// TIA Portal V16 export
// export: Created 2021-12-01T20:36:09.36916Z, ExportSetting WithDefaults, DisplayName Totally Integrated Automation Portal, DisplayVersion V16 Update 4, DisplayName TIA Portal Version Control Interface, DisplayVersion V16 Update 2, DisplayName TIA Portal Openness, DisplayVersion V16 Update 4, DisplayName SINAMICS Startdrive Advanced, DisplayVersion V16 Update 5, DisplayName SINAMICS Startdrive G130, G150, S120, S150, SINAMICS MV, S210, DisplayVersion V16 Update 5, DisplayName SINAMICS Startdrive G110M, G120, G120C, G120D, G120P, G115D, DisplayVersion V16 Update 5, DisplayName STEP 7 Professional, DisplayVersion V16 Update 4, DisplayName STEP 7 Safety, DisplayVersion V16, DisplayName WinCC Advanced, DisplayVersion V16 Update 4
FUNCTION "ST00310_FC" : Void   // FC42, LAD
TITLE = ST00310
{ S7_Optimized_Access := 'TRUE' }
VERSION : 0.1
// stored: AutoNumber true, IsIECCheckEnabled false, SetENOAutomatically false, UDAEnableTagReadback false
   VAR_IN_OUT
      OPMODE : "OPMODE_OUT_UDT";
      HMI_EXTENSION : "HMI_EXTENSION_PANEL_UDT";
   END_VAR
   VAR_TEMP
      VDL_TargetPosition : DInt;   // VDL - Target position
      VDL_StartPositioning : Bool;   // VDL - Start auto positioning
      Empty_HS : "RT_HANDSHAKE_UDT";
      PlantIdentifier : WString;
   END_VAR
   VAR CONSTANT
      GetPayloadUID : String := 'ST00310_GP';
   END_VAR
   VAR_TEMP   // added for the SCL form of the ladder/FBD networks
      _w1 : Bool;
      _w2 : Bool;
   END_VAR
BEGIN

REGION Network 1: Alarm
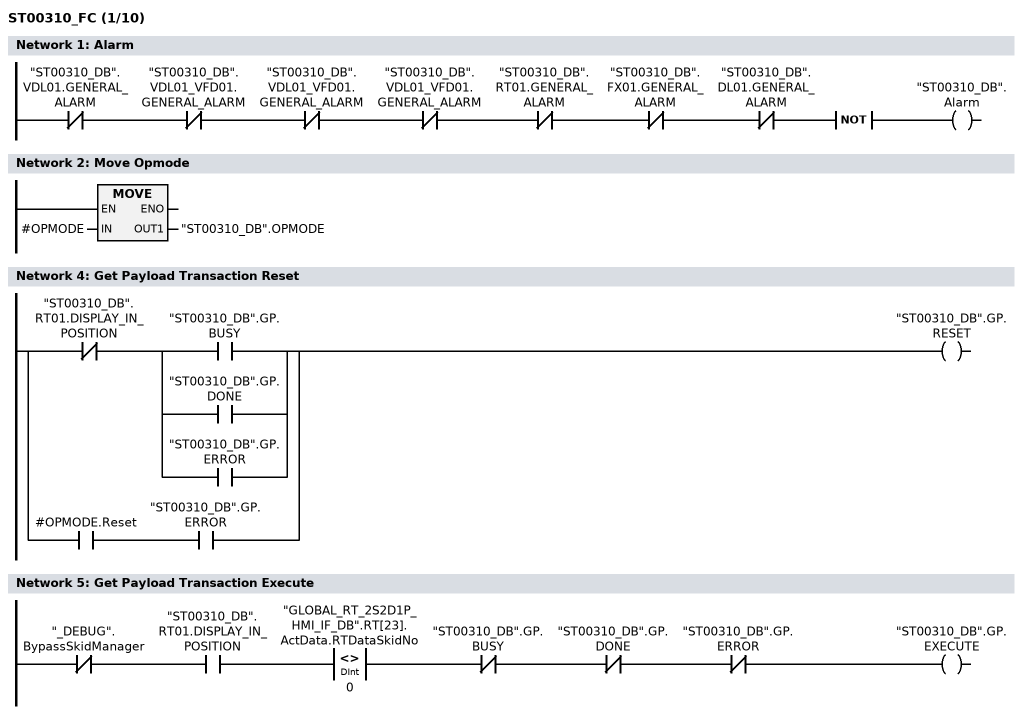
   RUNG wire#powerrail
      I_Contact( "ST00310_DB".VDL01.GENERAL_ALARM )
      I_Contact( "ST00310_DB".VDL01_VFD01.GENERAL_ALARM )
      I_Contact( "ST00310_DB".VDL01_VFD01.GENERAL_ALARM )
      I_Contact( "ST00310_DB".VDL01_VFD01.GENERAL_ALARM )
      I_Contact( "ST00310_DB".RT01.GENERAL_ALARM )
      I_Contact( "ST00310_DB".FX01.GENERAL_ALARM )
      I_Contact( "ST00310_DB".DL01.GENERAL_ALARM )
      Not()
      Coil( "ST00310_DB".Alarm )
   END_RUNG
   // the same network as SCL:
   "ST00310_DB".Alarm := NOT (NOT "ST00310_DB".VDL01.GENERAL_ALARM AND NOT "ST00310_DB".VDL01_VFD01.GENERAL_ALARM AND NOT "ST00310_DB".VDL01_VFD01.GENERAL_ALARM AND NOT "ST00310_DB".VDL01_VFD01.GENERAL_ALARM AND NOT "ST00310_DB".RT01.GENERAL_ALARM AND NOT "ST00310_DB".FX01.GENERAL_ALARM AND NOT "ST00310_DB".DL01.GENERAL_ALARM);
END_REGION

REGION Network 2: Move Opmode
   RUNG wire#powerrail
      Move(in := #OPMODE, out1 => "ST00310_DB".OPMODE)
   END_RUNG
   // the same network as SCL:
   "ST00310_DB".OPMODE := #OPMODE;
END_REGION

REGION Network 3: ==== Get Payload ====
END_REGION

REGION Network 4: Get Payload Transaction Reset
   RUNG wire#powerrail
      I_Contact( "ST00310_DB".RT01.DISPLAY_IN_POSITION )
      wire#w1
      Contact( "ST00310_DB".GP.BUSY )
      wire#w2
      Coil( "ST00310_DB".GP.RESET )
   END_RUNG
   RUNG wire#w1
      Contact( "ST00310_DB".GP.DONE )
   END_RUNG wire#w2
   RUNG wire#w1
      Contact( "ST00310_DB".GP.ERROR )
   END_RUNG wire#w2
   RUNG wire#powerrail
      Contact( #OPMODE.Reset )
      Contact( "ST00310_DB".GP.ERROR )
   END_RUNG wire#w2
   // the same network as SCL:
   "ST00310_DB".GP.RESET := (NOT "ST00310_DB".RT01.DISPLAY_IN_POSITION AND ("ST00310_DB".GP.BUSY OR "ST00310_DB".GP.DONE OR "ST00310_DB".GP.ERROR)) OR (#OPMODE.Reset AND "ST00310_DB".GP.ERROR);
END_REGION

REGION Network 5: Get Payload Transaction Execute
   RUNG wire#powerrail
      I_Contact( "_DEBUG".BypassSkidManager )
      Contact( "ST00310_DB".RT01.DISPLAY_IN_POSITION )
      { S7_Templates := "SrcType := DInt" } NE_Contact(in1 := "GLOBAL_RT_2S2D1P_HMI_IF_DB".RT[23].ActData.RTDataSkidNo, in2 := 0)
      I_Contact( "ST00310_DB".GP.BUSY )
      I_Contact( "ST00310_DB".GP.DONE )
      I_Contact( "ST00310_DB".GP.ERROR )
      Coil( "ST00310_DB".GP.EXECUTE )
   END_RUNG
   // the same network as SCL:
   "ST00310_DB".GP.EXECUTE := NOT "_DEBUG".BypassSkidManager AND "ST00310_DB".RT01.DISPLAY_IN_POSITION AND ("GLOBAL_RT_2S2D1P_HMI_IF_DB".RT[23].ActData.RTDataSkidNo <> 0) AND NOT "ST00310_DB".GP.BUSY AND NOT "ST00310_DB".GP.DONE AND NOT "ST00310_DB".GP.ERROR;
END_REGION

REGION Network 6: Get Payload Transaction Control
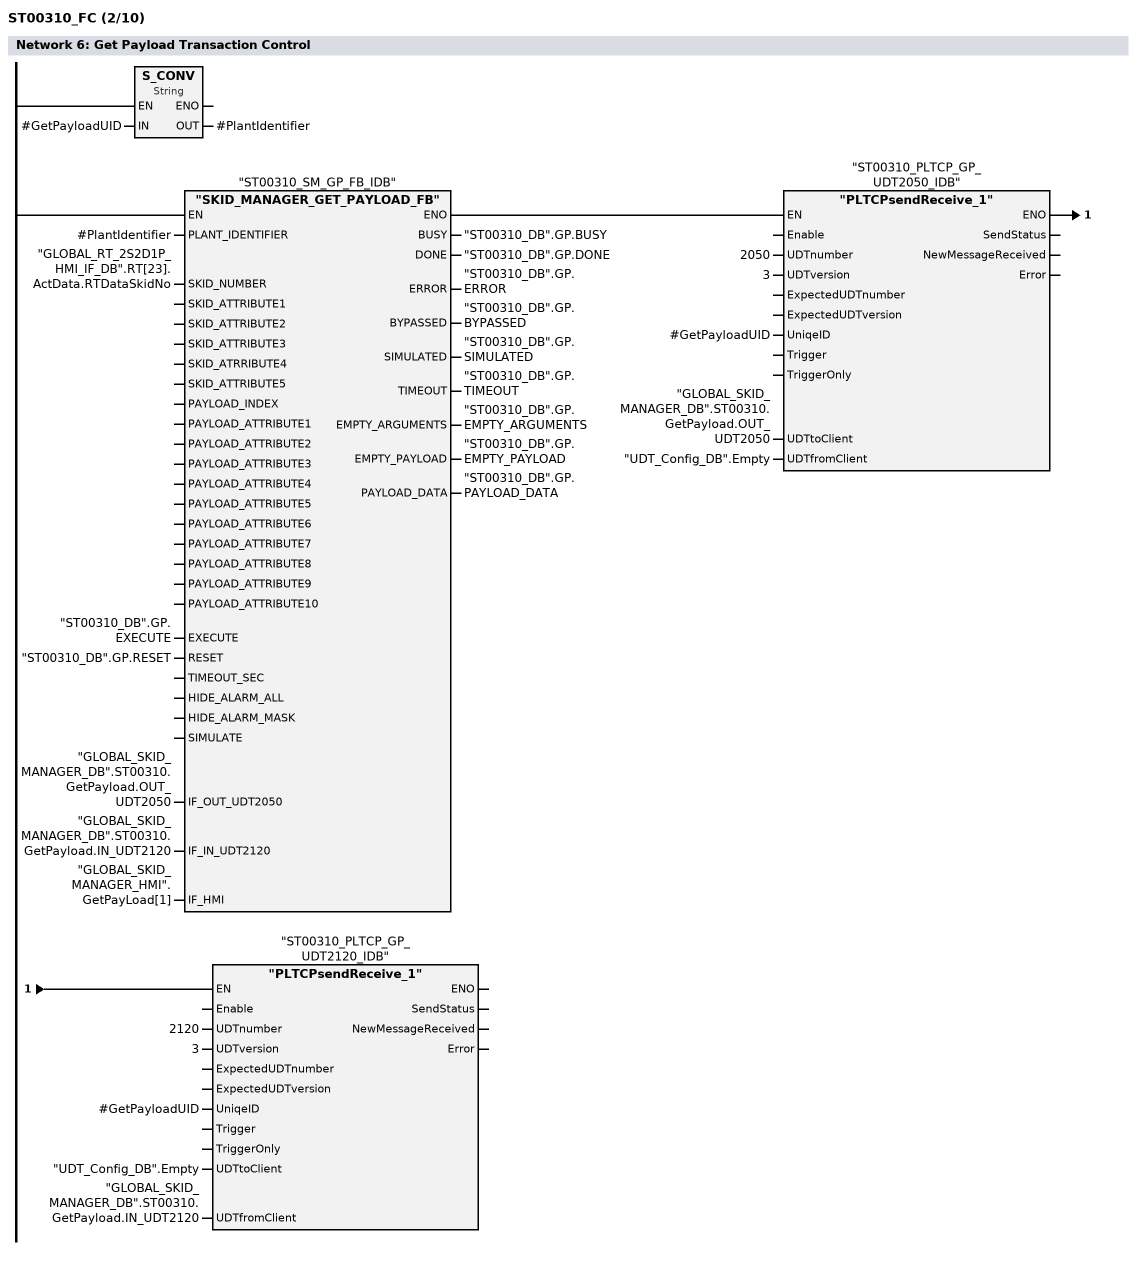
   RUNG wire#powerrail
      { S7_Templates := "[src_type := String, dest_type := WString]" } S_CONV(IN := #GetPayloadUID, OUT => #PlantIdentifier)
   END_RUNG
   RUNG wire#powerrail
      "ST00310_SM_GP_FB_IDB"(PLANT_IDENTIFIER := #PlantIdentifier, SKID_NUMBER := "GLOBAL_RT_2S2D1P_HMI_IF_DB".RT[23].ActData.RTDataSkidNo, SKID_ATTRIBUTE1 :=, SKID_ATTRIBUTE2 :=, SKID_ATTRIBUTE3 :=, SKID_ATRRIBUTE4 :=, SKID_ATTRIBUTE5 :=, PAYLOAD_INDEX :=, PAYLOAD_ATTRIBUTE1 :=, PAYLOAD_ATTRIBUTE2 :=, PAYLOAD_ATTRIBUTE3 :=, PAYLOAD_ATTRIBUTE4 :=, PAYLOAD_ATTRIBUTE5 :=, PAYLOAD_ATTRIBUTE6 :=, PAYLOAD_ATTRIBUTE7 :=, PAYLOAD_ATTRIBUTE8 :=, PAYLOAD_ATTRIBUTE9 :=, PAYLOAD_ATTRIBUTE10 :=, EXECUTE := "ST00310_DB".GP.EXECUTE, RESET := "ST00310_DB".GP.RESET, TIMEOUT_SEC :=, HIDE_ALARM_ALL :=, HIDE_ALARM_MASK :=, SIMULATE :=, IF_OUT_UDT2050 := "GLOBAL_SKID_MANAGER_DB".ST00310.GetPayload.OUT_UDT2050, IF_IN_UDT2120 := "GLOBAL_SKID_MANAGER_DB".ST00310.GetPayload.IN_UDT2120, IF_HMI := "GLOBAL_SKID_MANAGER_HMI".GetPayLoad[1], BUSY => "ST00310_DB".GP.BUSY, DONE => "ST00310_DB".GP.DONE, ERROR => "ST00310_DB".GP.ERROR, BYPASSED => "ST00310_DB".GP.BYPASSED, SIMULATED => "ST00310_DB".GP.SIMULATED, TIMEOUT => "ST00310_DB".GP.TIMEOUT, EMPTY_ARGUMENTS => "ST00310_DB".GP.EMPTY_ARGUMENTS, EMPTY_PAYLOAD => "ST00310_DB".GP.EMPTY_PAYLOAD, PAYLOAD_DATA => "ST00310_DB".GP.PAYLOAD_DATA)
      "ST00310_PLTCP_GP_UDT2050_IDB"(Enable :=, UDTnumber := 2050, UDTversion := 3, ExpectedUDTnumber :=, ExpectedUDTversion :=, UniqeID := #GetPayloadUID, Trigger :=, TriggerOnly :=, UDTtoClient := "GLOBAL_SKID_MANAGER_DB".ST00310.GetPayload.OUT_UDT2050, UDTfromClient := "UDT_Config_DB".Empty, SendStatus =>, NewMessageReceived =>, Error =>)
      "ST00310_PLTCP_GP_UDT2120_IDB"(Enable :=, UDTnumber := 2120, UDTversion := 3, ExpectedUDTnumber :=, ExpectedUDTversion :=, UniqeID := #GetPayloadUID, Trigger :=, TriggerOnly :=, UDTtoClient := "UDT_Config_DB".Empty, UDTfromClient := "GLOBAL_SKID_MANAGER_DB".ST00310.GetPayload.IN_UDT2120, SendStatus =>, NewMessageReceived =>, Error =>)
   END_RUNG
   // the same network as SCL:
   S_CONV(IN := #GetPayloadUID, OUT => #PlantIdentifier);
   "ST00310_SM_GP_FB_IDB"(PLANT_IDENTIFIER := #PlantIdentifier,   // "SKID_MANAGER_GET_PAYLOAD_FB"
                          SKID_NUMBER := "GLOBAL_RT_2S2D1P_HMI_IF_DB".RT[23].ActData.RTDataSkidNo,
                          EXECUTE := "ST00310_DB".GP.EXECUTE,
                          RESET := "ST00310_DB".GP.RESET,
                          IF_OUT_UDT2050 := "GLOBAL_SKID_MANAGER_DB".ST00310.GetPayload.OUT_UDT2050,
                          IF_IN_UDT2120 := "GLOBAL_SKID_MANAGER_DB".ST00310.GetPayload.IN_UDT2120,
                          IF_HMI := "GLOBAL_SKID_MANAGER_HMI".GetPayLoad[1],
                          BUSY => "ST00310_DB".GP.BUSY,
                          DONE => "ST00310_DB".GP.DONE,
                          ERROR => "ST00310_DB".GP.ERROR,
                          BYPASSED => "ST00310_DB".GP.BYPASSED,
                          SIMULATED => "ST00310_DB".GP.SIMULATED,
                          TIMEOUT => "ST00310_DB".GP.TIMEOUT,
                          EMPTY_ARGUMENTS => "ST00310_DB".GP.EMPTY_ARGUMENTS,
                          EMPTY_PAYLOAD => "ST00310_DB".GP.EMPTY_PAYLOAD,
                          PAYLOAD_DATA => "ST00310_DB".GP.PAYLOAD_DATA,
                          ENO => #_w1);
   "ST00310_PLTCP_GP_UDT2050_IDB"(EN := #_w1,   // "PLTCPsendReceive_1"
                           UDTnumber := 2050,
                           UDTversion := 3,
                           UniqeID := #GetPayloadUID,
                           UDTtoClient := "GLOBAL_SKID_MANAGER_DB".ST00310.GetPayload.OUT_UDT2050,
                           UDTfromClient := "UDT_Config_DB".Empty,
                           ENO => #_w2);
   IF #_w2 THEN
       "ST00310_PLTCP_GP_UDT2120_IDB"(UDTnumber := 2120,   // "PLTCPsendReceive_1"
                               UDTversion := 3,
                               UniqeID := #GetPayloadUID,
                               UDTtoClient := "UDT_Config_DB".Empty,
                               UDTfromClient := "GLOBAL_SKID_MANAGER_DB".ST00310.GetPayload.IN_UDT2120);
   END_IF;
END_REGION

REGION Network 7: *******************VDL01 Control*******************
END_REGION

REGION Network 8 (SCL): VDL01 Parameters


   "ST00310_DB".VDL01.PARA_SET.Para.StopNextPos := true;
   "ST00310_DB".VDL01.PARA_SET.Set.DistPos := 10;
   "ST00310_DB".VDL01.PARA_SET.Set.DistSDFwd := 550;
   "ST00310_DB".VDL01.PARA_SET.Set.DistSDRev := 550;
   "ST00310_DB".VDL01.PARA_SET.Set.DistStopFwd := 20;
   "ST00310_DB".VDL01.PARA_SET.Set.DistStopRev := 20;
   "ST00310_DB".VDL01.PARA_SET.Set.EncValFac := 1;
   "ST00310_DB".VDL01.PARA_SET.Set.LastPos := 2;
   "ST00310_DB".VDL01.PARA_SET.Set.LimSwSWFwd := 9130;
   "ST00310_DB".VDL01.PARA_SET.Set.LimSwSWRev := 550;


   "ST00310_DB".VDL01.PARA_SET.Set.Pos1S := 590;
   "ST00310_DB".VDL01.PARA_SET.Set.Pos2S := 9115;

   "ST00310_DB".VDL01.PARA_SET.Set.RtPos1Pos2 := 300;
END_REGION

REGION Network 9: VDL01 Distance Meter
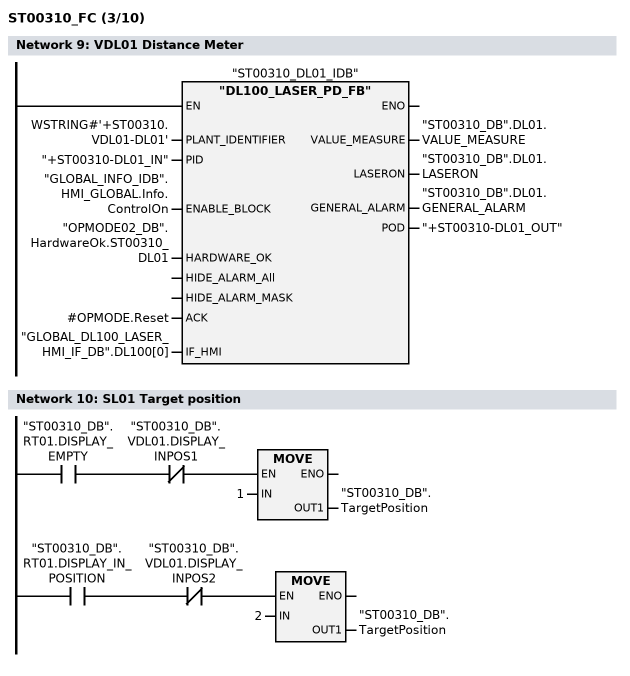
   RUNG wire#powerrail
      "ST00310_DL01_IDB"(PLANT_IDENTIFIER := WSTRING#'+ST00310.VDL01-DL01', PID := "+ST00310-DL01_IN", ENABLE_BLOCK := "GLOBAL_INFO_IDB".HMI_GLOBAL.Info.ControlOn, HARDWARE_OK := "OPMODE02_DB".HardwareOk.ST00310_DL01, HIDE_ALARM_All :=, HIDE_ALARM_MASK :=, ACK := #OPMODE.Reset, IF_HMI := "GLOBAL_DL100_LASER_HMI_IF_DB".DL100[0], VALUE_MEASURE => "ST00310_DB".DL01.VALUE_MEASURE, LASERON => "ST00310_DB".DL01.LASERON, GENERAL_ALARM => "ST00310_DB".DL01.GENERAL_ALARM, POD => "+ST00310-DL01_OUT")
   END_RUNG
   // the same network as SCL:
   "ST00310_DL01_IDB"(PLANT_IDENTIFIER := WSTRING#'+ST00310.VDL01-DL01',   // "DL100_LASER_PD_FB"
                      PID := "+ST00310-DL01_IN",
                      ENABLE_BLOCK := "GLOBAL_INFO_IDB".HMI_GLOBAL.Info.ControlOn,
                      HARDWARE_OK := "OPMODE02_DB".HardwareOk.ST00310_DL01,
                      ACK := #OPMODE.Reset,
                      IF_HMI := "GLOBAL_DL100_LASER_HMI_IF_DB".DL100[0],
                      VALUE_MEASURE => "ST00310_DB".DL01.VALUE_MEASURE,
                      LASERON => "ST00310_DB".DL01.LASERON,
                      GENERAL_ALARM => "ST00310_DB".DL01.GENERAL_ALARM,
                      POD => "+ST00310-DL01_OUT");
END_REGION

REGION Network 10: SL01 Target position
   RUNG wire#powerrail
      Contact( "ST00310_DB".RT01.DISPLAY_EMPTY )
      I_Contact( "ST00310_DB".VDL01.DISPLAY_INPOS1 )
      Move(in := 1, out1 => "ST00310_DB".TargetPosition)
   END_RUNG
   RUNG wire#powerrail
      Contact( "ST00310_DB".RT01.DISPLAY_IN_POSITION )
      I_Contact( "ST00310_DB".VDL01.DISPLAY_INPOS2 )
      Move(in := 2, out1 => "ST00310_DB".TargetPosition)
   END_RUNG
   // the same network as SCL:
   IF "ST00310_DB".RT01.DISPLAY_EMPTY AND NOT "ST00310_DB".VDL01.DISPLAY_INPOS1 THEN
       "ST00310_DB".TargetPosition := 1;
   END_IF;
   IF "ST00310_DB".RT01.DISPLAY_IN_POSITION AND NOT "ST00310_DB".VDL01.DISPLAY_INPOS2 THEN
       "ST00310_DB".TargetPosition := 2;
   END_IF;
END_REGION

REGION Network 11: VDL01 FB Control
   // 1. RT occupied -> go to 8,5m
   // 2. RT not occupied -> go to 0m
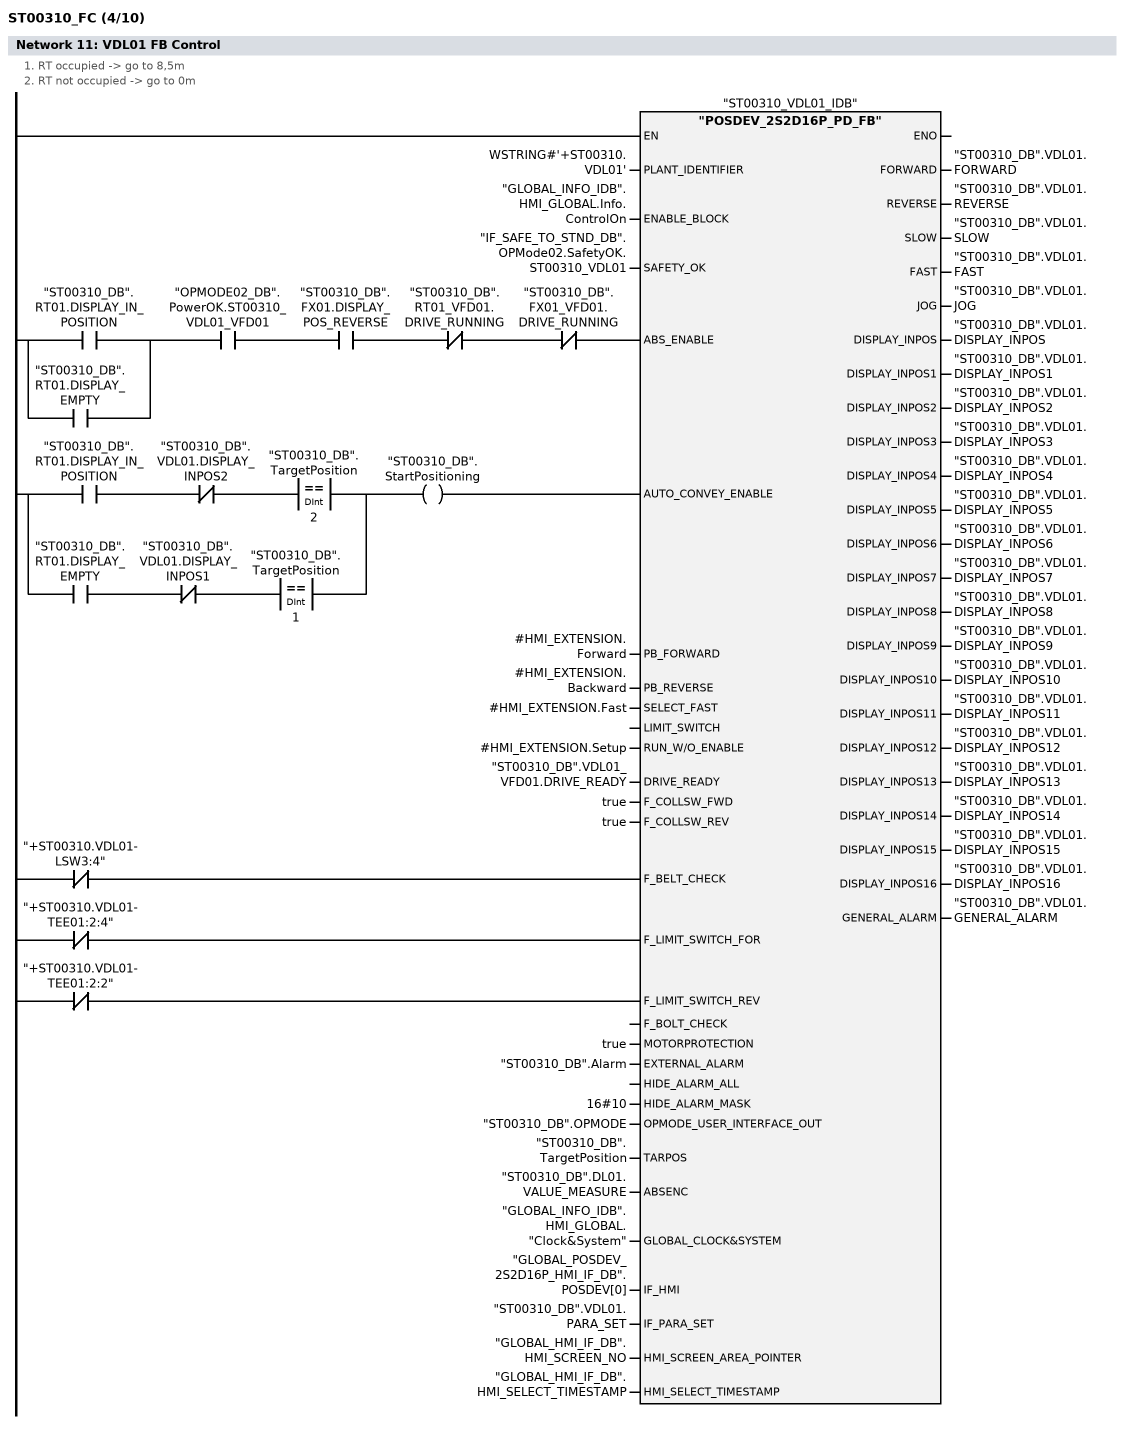
   RUNG wire#powerrail
      "ST00310_VDL01_IDB"(ABS_ENABLE := wire#w2, AUTO_CONVEY_ENABLE := wire#w4, F_BELT_CHECK := wire#w5, F_LIMIT_SWITCH_FOR := wire#w6, F_LIMIT_SWITCH_REV := wire#w7, PLANT_IDENTIFIER := WSTRING#'+ST00310.VDL01', ENABLE_BLOCK := "GLOBAL_INFO_IDB".HMI_GLOBAL.Info.ControlOn, SAFETY_OK := "IF_SAFE_TO_STND_DB".OPMode02.SafetyOK.ST00310_VDL01, PB_FORWARD := #HMI_EXTENSION.Forward, PB_REVERSE := #HMI_EXTENSION.Backward, SELECT_FAST := #HMI_EXTENSION.Fast, LIMIT_SWITCH :=, "RUN_W/O_ENABLE" := #HMI_EXTENSION.Setup, DRIVE_READY := "ST00310_DB".VDL01_VFD01.DRIVE_READY, F_COLLSW_FWD := true, F_COLLSW_REV := true, F_BOLT_CHECK :=, MOTORPROTECTION := true, EXTERNAL_ALARM := "ST00310_DB".Alarm, HIDE_ALARM_ALL :=, HIDE_ALARM_MASK := 16#10, OPMODE_USER_INTERFACE_OUT := "ST00310_DB".OPMODE, TARPOS := "ST00310_DB".TargetPosition, ABSENC := "ST00310_DB".DL01.VALUE_MEASURE, "GLOBAL_CLOCK&SYSTEM" := "GLOBAL_INFO_IDB".HMI_GLOBAL."Clock&System", IF_HMI := "GLOBAL_POSDEV_2S2D16P_HMI_IF_DB".POSDEV[0], IF_PARA_SET := "ST00310_DB".VDL01.PARA_SET, HMI_SCREEN_AREA_POINTER := "GLOBAL_HMI_IF_DB".HMI_SCREEN_NO, HMI_SELECT_TIMESTAMP := "GLOBAL_HMI_IF_DB".HMI_SELECT_TIMESTAMP, FORWARD => "ST00310_DB".VDL01.FORWARD, REVERSE => "ST00310_DB".VDL01.REVERSE, SLOW => "ST00310_DB".VDL01.SLOW, FAST => "ST00310_DB".VDL01.FAST, JOG => "ST00310_DB".VDL01.JOG, DISPLAY_INPOS => "ST00310_DB".VDL01.DISPLAY_INPOS, DISPLAY_INPOS1 => "ST00310_DB".VDL01.DISPLAY_INPOS1, DISPLAY_INPOS2 => "ST00310_DB".VDL01.DISPLAY_INPOS2, DISPLAY_INPOS3 => "ST00310_DB".VDL01.DISPLAY_INPOS3, DISPLAY_INPOS4 => "ST00310_DB".VDL01.DISPLAY_INPOS4, DISPLAY_INPOS5 => "ST00310_DB".VDL01.DISPLAY_INPOS5, DISPLAY_INPOS6 => "ST00310_DB".VDL01.DISPLAY_INPOS6, DISPLAY_INPOS7 => "ST00310_DB".VDL01.DISPLAY_INPOS7, DISPLAY_INPOS8 => "ST00310_DB".VDL01.DISPLAY_INPOS8, DISPLAY_INPOS9 => "ST00310_DB".VDL01.DISPLAY_INPOS9, DISPLAY_INPOS10 => "ST00310_DB".VDL01.DISPLAY_INPOS10, DISPLAY_INPOS11 => "ST00310_DB".VDL01.DISPLAY_INPOS11, DISPLAY_INPOS12 => "ST00310_DB".VDL01.DISPLAY_INPOS12, DISPLAY_INPOS13 => "ST00310_DB".VDL01.DISPLAY_INPOS13, DISPLAY_INPOS14 => "ST00310_DB".VDL01.DISPLAY_INPOS14, DISPLAY_INPOS15 => "ST00310_DB".VDL01.DISPLAY_INPOS15, DISPLAY_INPOS16 => "ST00310_DB".VDL01.DISPLAY_INPOS16, GENERAL_ALARM => "ST00310_DB".VDL01.GENERAL_ALARM)
   END_RUNG
   RUNG wire#powerrail
      Contact( "ST00310_DB".RT01.DISPLAY_IN_POSITION )
      wire#w1
      Contact( "OPMODE02_DB".PowerOK.ST00310_VDL01_VFD01 )
      Contact( "ST00310_DB".FX01.DISPLAY_POS_REVERSE )
      I_Contact( "ST00310_DB".RT01_VFD01.DRIVE_RUNNING )
      I_Contact( "ST00310_DB".FX01_VFD01.DRIVE_RUNNING )
   END_RUNG wire#w2
   RUNG wire#powerrail
      Contact( "ST00310_DB".RT01.DISPLAY_EMPTY )
   END_RUNG wire#w1
   RUNG wire#powerrail
      Contact( "ST00310_DB".RT01.DISPLAY_IN_POSITION )
      I_Contact( "ST00310_DB".VDL01.DISPLAY_INPOS2 )
      { S7_Templates := "SrcType := DInt" } EQ_Contact(in1 := "ST00310_DB".TargetPosition, in2 := 2)
      wire#w3
      Coil( "ST00310_DB".StartPositioning )
   END_RUNG wire#w4
   RUNG wire#powerrail
      Contact( "ST00310_DB".RT01.DISPLAY_EMPTY )
      I_Contact( "ST00310_DB".VDL01.DISPLAY_INPOS1 )
      { S7_Templates := "SrcType := DInt" } EQ_Contact(in1 := "ST00310_DB".TargetPosition, in2 := 1)
   END_RUNG wire#w3
   RUNG wire#powerrail
      I_Contact( "+ST00310.VDL01-LSW3:4" )
   END_RUNG wire#w5
   RUNG wire#powerrail
      I_Contact( "+ST00310.VDL01-TEE01:2:4" )
   END_RUNG wire#w6
   RUNG wire#powerrail
      I_Contact( "+ST00310.VDL01-TEE01:2:2" )
   END_RUNG wire#w7
   // the same network as SCL:
   "ST00310_DB".StartPositioning := ("ST00310_DB".RT01.DISPLAY_IN_POSITION AND NOT "ST00310_DB".VDL01.DISPLAY_INPOS2 AND ("ST00310_DB".TargetPosition = 2)) OR ("ST00310_DB".RT01.DISPLAY_EMPTY AND NOT "ST00310_DB".VDL01.DISPLAY_INPOS1 AND ("ST00310_DB".TargetPosition = 1));
   "ST00310_VDL01_IDB"(PLANT_IDENTIFIER := WSTRING#'+ST00310.VDL01',   // "POSDEV_2S2D16P_PD_FB"
                       ENABLE_BLOCK := "GLOBAL_INFO_IDB".HMI_GLOBAL.Info.ControlOn,
                       SAFETY_OK := "IF_SAFE_TO_STND_DB".OPMode02.SafetyOK.ST00310_VDL01,
                       ABS_ENABLE := ("ST00310_DB".RT01.DISPLAY_IN_POSITION OR "ST00310_DB".RT01.DISPLAY_EMPTY) AND "OPMODE02_DB".PowerOK.ST00310_VDL01_VFD01 AND "ST00310_DB".FX01.DISPLAY_POS_REVERSE AND NOT "ST00310_DB".RT01_VFD01.DRIVE_RUNNING AND NOT "ST00310_DB".FX01_VFD01.DRIVE_RUNNING,
                       AUTO_CONVEY_ENABLE := "ST00310_DB".StartPositioning,
                       PB_FORWARD := #HMI_EXTENSION.Forward,
                       PB_REVERSE := #HMI_EXTENSION.Backward,
                       SELECT_FAST := #HMI_EXTENSION.Fast,
                       "RUN_W/O_ENABLE" := #HMI_EXTENSION.Setup,
                       DRIVE_READY := "ST00310_DB".VDL01_VFD01.DRIVE_READY,
                       F_COLLSW_FWD := true,
                       F_COLLSW_REV := true,
                       F_BELT_CHECK := NOT "+ST00310.VDL01-LSW3:4",
                       F_LIMIT_SWITCH_FOR := NOT "+ST00310.VDL01-TEE01:2:4",
                       F_LIMIT_SWITCH_REV := NOT "+ST00310.VDL01-TEE01:2:2",
                       MOTORPROTECTION := true,
                       EXTERNAL_ALARM := "ST00310_DB".Alarm,
                       HIDE_ALARM_MASK := 16#10,
                       OPMODE_USER_INTERFACE_OUT := "ST00310_DB".OPMODE,
                       TARPOS := "ST00310_DB".TargetPosition,
                       ABSENC := "ST00310_DB".DL01.VALUE_MEASURE,
                       "GLOBAL_CLOCK&SYSTEM" := "GLOBAL_INFO_IDB".HMI_GLOBAL."Clock&System",
                       IF_HMI := "GLOBAL_POSDEV_2S2D16P_HMI_IF_DB".POSDEV[0],
                       IF_PARA_SET := "ST00310_DB".VDL01.PARA_SET,
                       HMI_SCREEN_AREA_POINTER := "GLOBAL_HMI_IF_DB".HMI_SCREEN_NO,
                       HMI_SELECT_TIMESTAMP := "GLOBAL_HMI_IF_DB".HMI_SELECT_TIMESTAMP,
                       FORWARD => "ST00310_DB".VDL01.FORWARD,
                       REVERSE => "ST00310_DB".VDL01.REVERSE,
                       SLOW => "ST00310_DB".VDL01.SLOW,
                       FAST => "ST00310_DB".VDL01.FAST,
                       JOG => "ST00310_DB".VDL01.JOG,
                       DISPLAY_INPOS => "ST00310_DB".VDL01.DISPLAY_INPOS,
                       DISPLAY_INPOS1 => "ST00310_DB".VDL01.DISPLAY_INPOS1,
                       DISPLAY_INPOS2 => "ST00310_DB".VDL01.DISPLAY_INPOS2,
                       DISPLAY_INPOS3 => "ST00310_DB".VDL01.DISPLAY_INPOS3,
                       DISPLAY_INPOS4 => "ST00310_DB".VDL01.DISPLAY_INPOS4,
                       DISPLAY_INPOS5 => "ST00310_DB".VDL01.DISPLAY_INPOS5,
                       DISPLAY_INPOS6 => "ST00310_DB".VDL01.DISPLAY_INPOS6,
                       DISPLAY_INPOS7 => "ST00310_DB".VDL01.DISPLAY_INPOS7,
                       DISPLAY_INPOS8 => "ST00310_DB".VDL01.DISPLAY_INPOS8,
                       DISPLAY_INPOS9 => "ST00310_DB".VDL01.DISPLAY_INPOS9,
                       DISPLAY_INPOS10 => "ST00310_DB".VDL01.DISPLAY_INPOS10,
                       DISPLAY_INPOS11 => "ST00310_DB".VDL01.DISPLAY_INPOS11,
                       DISPLAY_INPOS12 => "ST00310_DB".VDL01.DISPLAY_INPOS12,
                       DISPLAY_INPOS13 => "ST00310_DB".VDL01.DISPLAY_INPOS13,
                       DISPLAY_INPOS14 => "ST00310_DB".VDL01.DISPLAY_INPOS14,
                       DISPLAY_INPOS15 => "ST00310_DB".VDL01.DISPLAY_INPOS15,
                       DISPLAY_INPOS16 => "ST00310_DB".VDL01.DISPLAY_INPOS16,
                       GENERAL_ALARM => "ST00310_DB".VDL01.GENERAL_ALARM);
END_REGION

REGION Network 12: VDL01 Speed
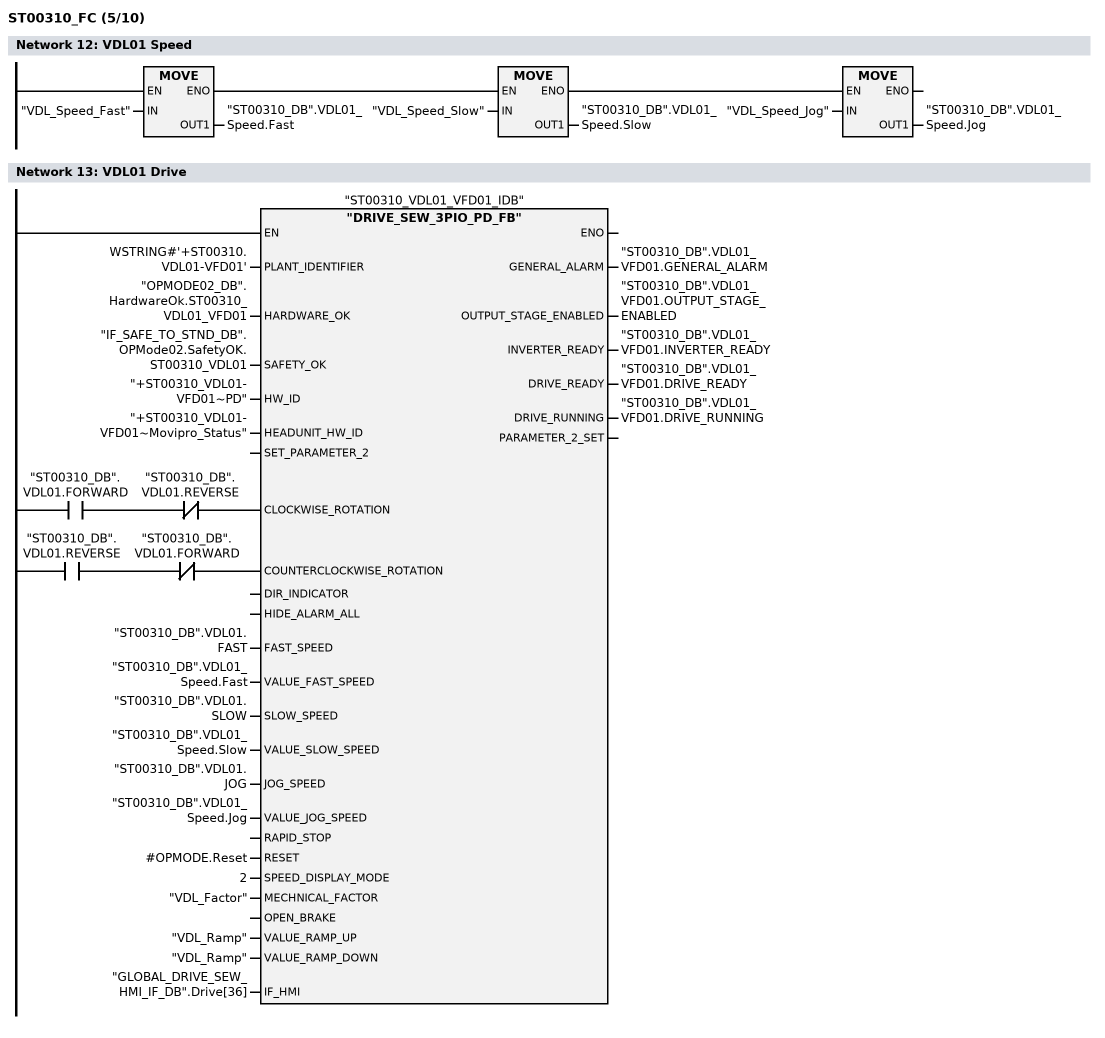
   RUNG wire#powerrail
      Move(in := "VDL_Speed_Fast", out1 => "ST00310_DB".VDL01_Speed.Fast)
      Move(in := "VDL_Speed_Slow", out1 => "ST00310_DB".VDL01_Speed.Slow)
      Move(in := "VDL_Speed_Jog", out1 => "ST00310_DB".VDL01_Speed.Jog)
   END_RUNG
   // the same network as SCL:
   "ST00310_DB".VDL01_Speed.Fast := "VDL_Speed_Fast";
   "ST00310_DB".VDL01_Speed.Slow := "VDL_Speed_Slow";
   "ST00310_DB".VDL01_Speed.Jog := "VDL_Speed_Jog";
END_REGION

REGION Network 13: VDL01 Drive
   RUNG wire#powerrail
      "ST00310_VDL01_VFD01_IDB"(CLOCKWISE_ROTATION := wire#w1, COUNTERCLOCKWISE_ROTATION := wire#w2, PLANT_IDENTIFIER := WSTRING#'+ST00310.VDL01-VFD01', HARDWARE_OK := "OPMODE02_DB".HardwareOk.ST00310_VDL01_VFD01, SAFETY_OK := "IF_SAFE_TO_STND_DB".OPMode02.SafetyOK.ST00310_VDL01, HW_ID := "+ST00310_VDL01-VFD01~PD", HEADUNIT_HW_ID := "+ST00310_VDL01-VFD01~Movipro_Status", SET_PARAMETER_2 :=, DIR_INDICATOR :=, HIDE_ALARM_ALL :=, FAST_SPEED := "ST00310_DB".VDL01.FAST, VALUE_FAST_SPEED := "ST00310_DB".VDL01_Speed.Fast, SLOW_SPEED := "ST00310_DB".VDL01.SLOW, VALUE_SLOW_SPEED := "ST00310_DB".VDL01_Speed.Slow, JOG_SPEED := "ST00310_DB".VDL01.JOG, VALUE_JOG_SPEED := "ST00310_DB".VDL01_Speed.Jog, RAPID_STOP :=, RESET := #OPMODE.Reset, SPEED_DISPLAY_MODE := 2, MECHNICAL_FACTOR := "VDL_Factor", OPEN_BRAKE :=, VALUE_RAMP_UP := "VDL_Ramp", VALUE_RAMP_DOWN := "VDL_Ramp", IF_HMI := "GLOBAL_DRIVE_SEW_HMI_IF_DB".Drive[36], GENERAL_ALARM => "ST00310_DB".VDL01_VFD01.GENERAL_ALARM, OUTPUT_STAGE_ENABLED => "ST00310_DB".VDL01_VFD01.OUTPUT_STAGE_ENABLED, INVERTER_READY => "ST00310_DB".VDL01_VFD01.INVERTER_READY, DRIVE_READY => "ST00310_DB".VDL01_VFD01.DRIVE_READY, DRIVE_RUNNING => "ST00310_DB".VDL01_VFD01.DRIVE_RUNNING, PARAMETER_2_SET =>)
   END_RUNG
   RUNG wire#powerrail
      Contact( "ST00310_DB".VDL01.FORWARD )
      I_Contact( "ST00310_DB".VDL01.REVERSE )
   END_RUNG wire#w1
   RUNG wire#powerrail
      Contact( "ST00310_DB".VDL01.REVERSE )
      I_Contact( "ST00310_DB".VDL01.FORWARD )
   END_RUNG wire#w2
   // the same network as SCL:
   "ST00310_VDL01_VFD01_IDB"(PLANT_IDENTIFIER := WSTRING#'+ST00310.VDL01-VFD01',   // "DRIVE_SEW_3PIO_PD_FB"
                           HARDWARE_OK := "OPMODE02_DB".HardwareOk.ST00310_VDL01_VFD01,
                           SAFETY_OK := "IF_SAFE_TO_STND_DB".OPMode02.SafetyOK.ST00310_VDL01,
                           HW_ID := "+ST00310_VDL01-VFD01~PD",
                           HEADUNIT_HW_ID := "+ST00310_VDL01-VFD01~Movipro_Status",
                           CLOCKWISE_ROTATION := "ST00310_DB".VDL01.FORWARD AND NOT "ST00310_DB".VDL01.REVERSE,
                           COUNTERCLOCKWISE_ROTATION := "ST00310_DB".VDL01.REVERSE AND NOT "ST00310_DB".VDL01.FORWARD,
                           FAST_SPEED := "ST00310_DB".VDL01.FAST,
                           VALUE_FAST_SPEED := "ST00310_DB".VDL01_Speed.Fast,
                           SLOW_SPEED := "ST00310_DB".VDL01.SLOW,
                           VALUE_SLOW_SPEED := "ST00310_DB".VDL01_Speed.Slow,
                           JOG_SPEED := "ST00310_DB".VDL01.JOG,
                           VALUE_JOG_SPEED := "ST00310_DB".VDL01_Speed.Jog,
                           RESET := #OPMODE.Reset,
                           SPEED_DISPLAY_MODE := 2,
                           MECHNICAL_FACTOR := "VDL_Factor",
                           VALUE_RAMP_UP := "VDL_Ramp",
                           VALUE_RAMP_DOWN := "VDL_Ramp",
                           IF_HMI := "GLOBAL_DRIVE_SEW_HMI_IF_DB".Drive[36],
                           GENERAL_ALARM => "ST00310_DB".VDL01_VFD01.GENERAL_ALARM,
                           OUTPUT_STAGE_ENABLED => "ST00310_DB".VDL01_VFD01.OUTPUT_STAGE_ENABLED,
                           INVERTER_READY => "ST00310_DB".VDL01_VFD01.INVERTER_READY,
                           DRIVE_READY => "ST00310_DB".VDL01_VFD01.DRIVE_READY,
                           DRIVE_RUNNING => "ST00310_DB".VDL01_VFD01.DRIVE_RUNNING);
END_REGION

REGION Network 14: *******************RT01 Control*******************
END_REGION

REGION Network 15 (SCL): RT01 Parameters
   "ST00310_DB".RT01.PARA_SET.Para.PosEndForward1 := true;
   "ST00310_DB".RT01.PARA_SET.Para.PosEndReverse := true;
   "ST00310_DB".RT01.PARA_SET.Para.PosSlowForward := true;
   "ST00310_DB".RT01.PARA_SET.Para.PosSlowReverse := false;
   "ST00310_DB".RT01.PARA_SET.Para.GapControlForward := false;
   "ST00310_DB".RT01.PARA_SET.Para.GapControlReverse := false;
   "ST00310_DB".RT01.PARA_SET.Para.NoStopTrans := true;
   "ST00310_DB".RT01.PARA_SET.Set.RunTimeForward := 450;
   "ST00310_DB".RT01.PARA_SET.Set.RunTimeReverse := 450;
END_REGION

REGION Network 16: RT01 HandShake
   // To do:
   // - Couple RT on 0m level
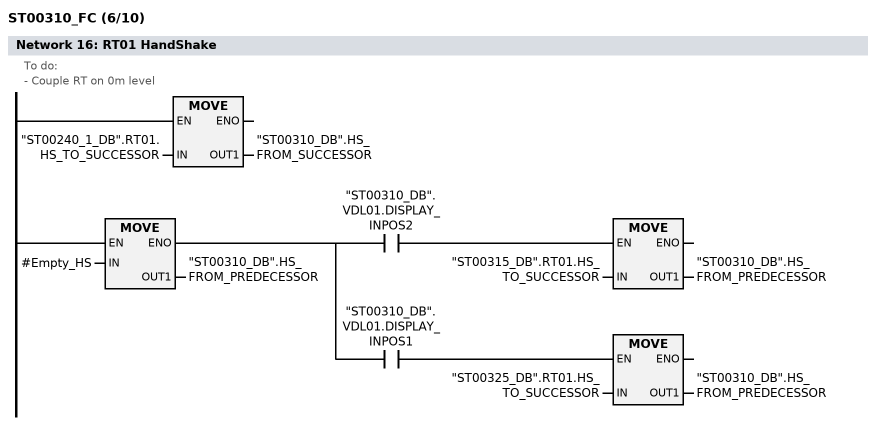
   RUNG wire#powerrail
      Move(in := "ST00240_1_DB".RT01.HS_TO_SUCCESSOR, out1 => "ST00310_DB".HS_FROM_SUCCESSOR)
   END_RUNG
   RUNG wire#powerrail
      Move(in := #Empty_HS, out1 => "ST00310_DB".HS_FROM_PREDECESSOR)
      wire#w1
      Contact( "ST00310_DB".VDL01.DISPLAY_INPOS2 )
      Move(in := "ST00315_DB".RT01.HS_TO_SUCCESSOR, out1 => "ST00310_DB".HS_FROM_PREDECESSOR)
   END_RUNG
   RUNG wire#w1
      Contact( "ST00310_DB".VDL01.DISPLAY_INPOS1 )
      Move(in := "ST00325_DB".RT01.HS_TO_SUCCESSOR, out1 => "ST00310_DB".HS_FROM_PREDECESSOR)
   END_RUNG
   // the same network as SCL:
   "ST00310_DB".HS_FROM_SUCCESSOR := "ST00240_1_DB".RT01.HS_TO_SUCCESSOR;
   "ST00310_DB".HS_FROM_PREDECESSOR := #Empty_HS;
   IF "ST00310_DB".VDL01.DISPLAY_INPOS2 THEN
       "ST00310_DB".HS_FROM_PREDECESSOR := "ST00315_DB".RT01.HS_TO_SUCCESSOR;
   END_IF;
   IF "ST00310_DB".VDL01.DISPLAY_INPOS1 THEN
       "ST00310_DB".HS_FROM_PREDECESSOR := "ST00325_DB".RT01.HS_TO_SUCCESSOR;
   END_IF;
END_REGION

REGION Network 17: RT01 FB Control
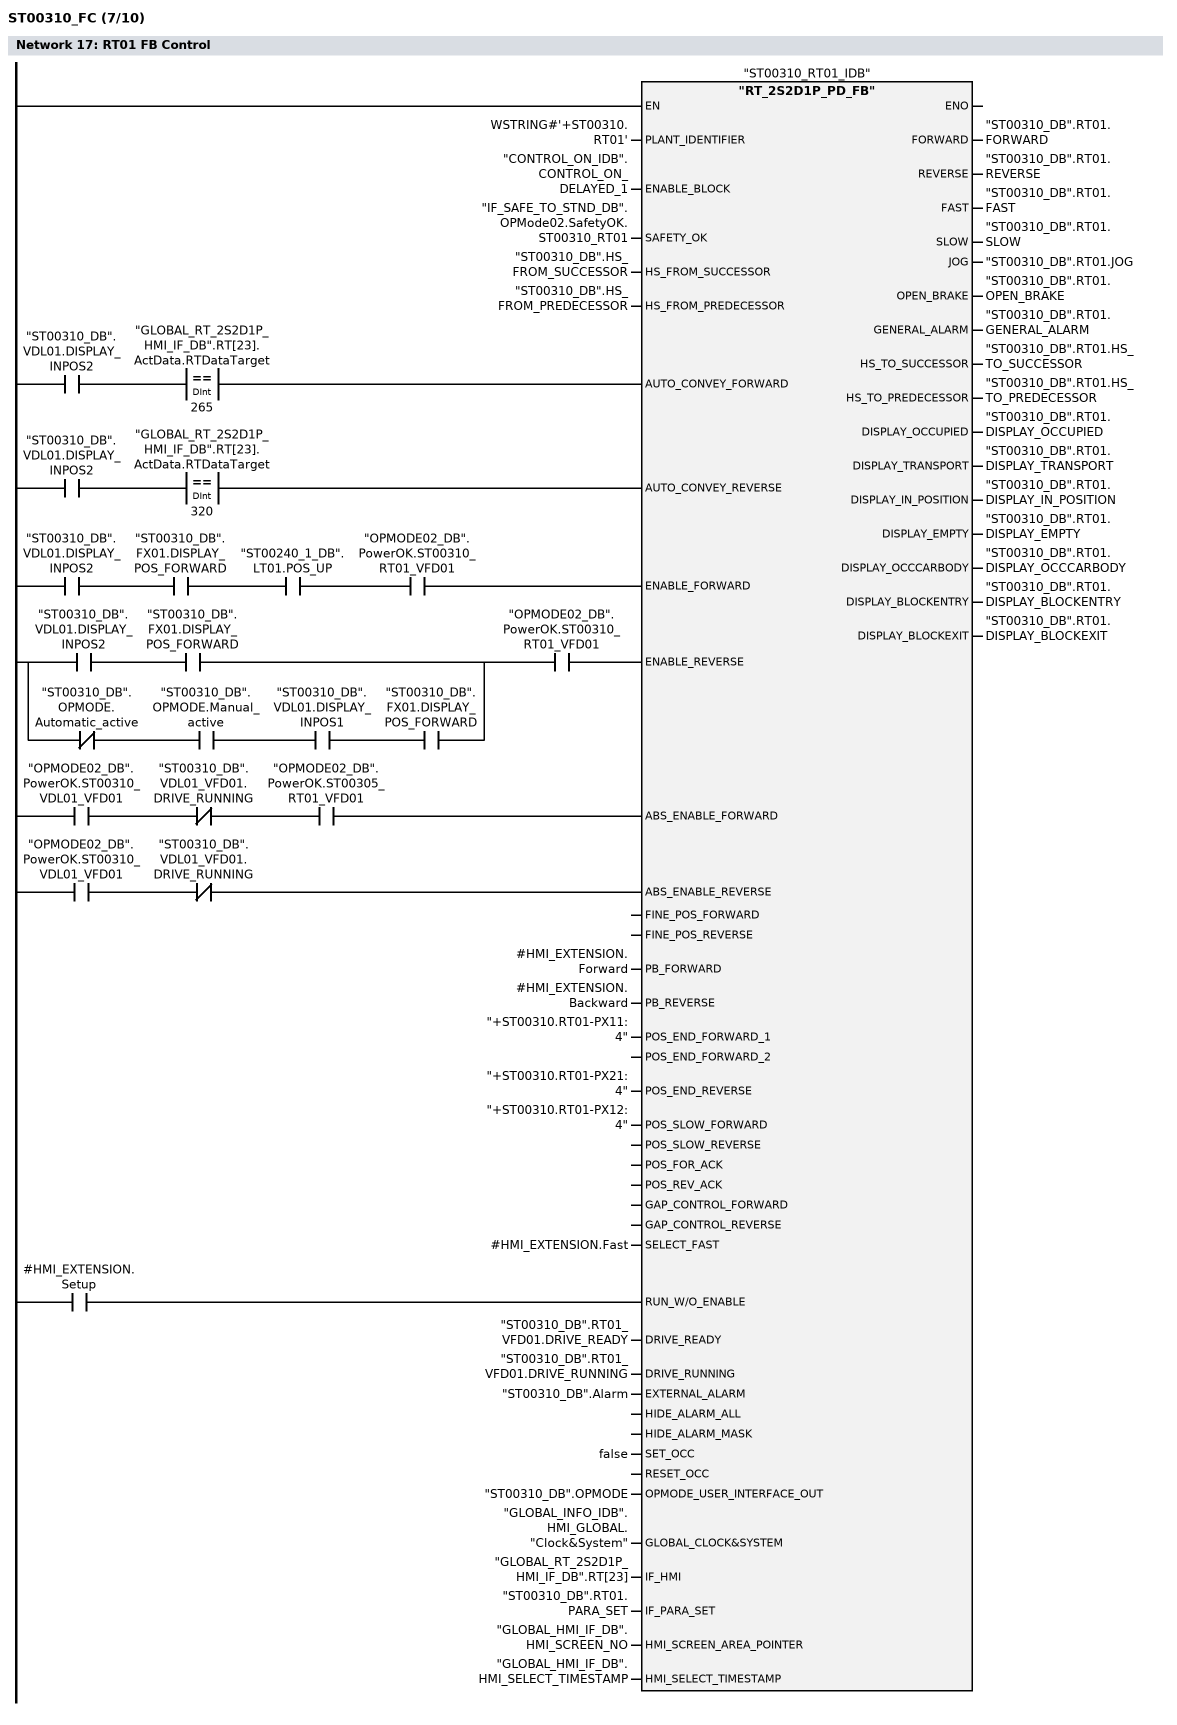
   RUNG wire#powerrail
      "ST00310_RT01_IDB"(AUTO_CONVEY_FORWARD := wire#w1, AUTO_CONVEY_REVERSE := wire#w2, ENABLE_FORWARD := wire#w3, ENABLE_REVERSE := wire#w5, ABS_ENABLE_FORWARD := wire#w6, ABS_ENABLE_REVERSE := wire#w7, "RUN_W/O_ENABLE" := wire#w8, PLANT_IDENTIFIER := WSTRING#'+ST00310.RT01', ENABLE_BLOCK := "CONTROL_ON_IDB".CONTROL_ON_DELAYED_1, SAFETY_OK := "IF_SAFE_TO_STND_DB".OPMode02.SafetyOK.ST00310_RT01, HS_FROM_SUCCESSOR := "ST00310_DB".HS_FROM_SUCCESSOR, HS_FROM_PREDECESSOR := "ST00310_DB".HS_FROM_PREDECESSOR, FINE_POS_FORWARD :=, FINE_POS_REVERSE :=, PB_FORWARD := #HMI_EXTENSION.Forward, PB_REVERSE := #HMI_EXTENSION.Backward, POS_END_FORWARD_1 := "+ST00310.RT01-PX11:4", POS_END_FORWARD_2 :=, POS_END_REVERSE := "+ST00310.RT01-PX21:4", POS_SLOW_FORWARD := "+ST00310.RT01-PX12:4", POS_SLOW_REVERSE :=, POS_FOR_ACK :=, POS_REV_ACK :=, GAP_CONTROL_FORWARD :=, GAP_CONTROL_REVERSE :=, SELECT_FAST := #HMI_EXTENSION.Fast, DRIVE_READY := "ST00310_DB".RT01_VFD01.DRIVE_READY, DRIVE_RUNNING := "ST00310_DB".RT01_VFD01.DRIVE_RUNNING, EXTERNAL_ALARM := "ST00310_DB".Alarm, HIDE_ALARM_ALL :=, HIDE_ALARM_MASK :=, SET_OCC := false, RESET_OCC :=, OPMODE_USER_INTERFACE_OUT := "ST00310_DB".OPMODE, "GLOBAL_CLOCK&SYSTEM" := "GLOBAL_INFO_IDB".HMI_GLOBAL."Clock&System", IF_HMI := "GLOBAL_RT_2S2D1P_HMI_IF_DB".RT[23], IF_PARA_SET := "ST00310_DB".RT01.PARA_SET, HMI_SCREEN_AREA_POINTER := "GLOBAL_HMI_IF_DB".HMI_SCREEN_NO, HMI_SELECT_TIMESTAMP := "GLOBAL_HMI_IF_DB".HMI_SELECT_TIMESTAMP, FORWARD => "ST00310_DB".RT01.FORWARD, REVERSE => "ST00310_DB".RT01.REVERSE, FAST => "ST00310_DB".RT01.FAST, SLOW => "ST00310_DB".RT01.SLOW, JOG => "ST00310_DB".RT01.JOG, OPEN_BRAKE => "ST00310_DB".RT01.OPEN_BRAKE, GENERAL_ALARM => "ST00310_DB".RT01.GENERAL_ALARM, HS_TO_SUCCESSOR => "ST00310_DB".RT01.HS_TO_SUCCESSOR, HS_TO_PREDECESSOR => "ST00310_DB".RT01.HS_TO_PREDECESSOR, DISPLAY_OCCUPIED => "ST00310_DB".RT01.DISPLAY_OCCUPIED, DISPLAY_TRANSPORT => "ST00310_DB".RT01.DISPLAY_TRANSPORT, DISPLAY_IN_POSITION => "ST00310_DB".RT01.DISPLAY_IN_POSITION, DISPLAY_EMPTY => "ST00310_DB".RT01.DISPLAY_EMPTY, DISPLAY_OCCCARBODY => "ST00310_DB".RT01.DISPLAY_OCCCARBODY, DISPLAY_BLOCKENTRY => "ST00310_DB".RT01.DISPLAY_BLOCKENTRY, DISPLAY_BLOCKEXIT => "ST00310_DB".RT01.DISPLAY_BLOCKEXIT)
   END_RUNG
   RUNG wire#powerrail
      Contact( "ST00310_DB".VDL01.DISPLAY_INPOS2 )
      { S7_Templates := "SrcType := DInt" } EQ_Contact(in1 := "GLOBAL_RT_2S2D1P_HMI_IF_DB".RT[23].ActData.RTDataTarget, in2 := 265)
   END_RUNG wire#w1
   RUNG wire#powerrail
      Contact( "ST00310_DB".VDL01.DISPLAY_INPOS2 )
      { S7_Templates := "SrcType := DInt" } EQ_Contact(in1 := "GLOBAL_RT_2S2D1P_HMI_IF_DB".RT[23].ActData.RTDataTarget, in2 := 320)
   END_RUNG wire#w2
   RUNG wire#powerrail
      Contact( "ST00310_DB".VDL01.DISPLAY_INPOS2 )
      Contact( "ST00310_DB".FX01.DISPLAY_POS_FORWARD )
      Contact( "ST00240_1_DB".LT01.POS_UP )
      Contact( "OPMODE02_DB".PowerOK.ST00310_RT01_VFD01 )
   END_RUNG wire#w3
   RUNG wire#powerrail
      Contact( "ST00310_DB".VDL01.DISPLAY_INPOS2 )
      Contact( "ST00310_DB".FX01.DISPLAY_POS_FORWARD )
      wire#w4
      Contact( "OPMODE02_DB".PowerOK.ST00310_RT01_VFD01 )
   END_RUNG wire#w5
   RUNG wire#powerrail
      I_Contact( "ST00310_DB".OPMODE.Automatic_active )
      Contact( "ST00310_DB".OPMODE.Manual_active )
      Contact( "ST00310_DB".VDL01.DISPLAY_INPOS1 )
      Contact( "ST00310_DB".FX01.DISPLAY_POS_FORWARD )
   END_RUNG wire#w4
   RUNG wire#powerrail
      Contact( "OPMODE02_DB".PowerOK.ST00310_VDL01_VFD01 )
      I_Contact( "ST00310_DB".VDL01_VFD01.DRIVE_RUNNING )
      Contact( "OPMODE02_DB".PowerOK.ST00305_RT01_VFD01 )
   END_RUNG wire#w6
   RUNG wire#powerrail
      Contact( "OPMODE02_DB".PowerOK.ST00310_VDL01_VFD01 )
      I_Contact( "ST00310_DB".VDL01_VFD01.DRIVE_RUNNING )
   END_RUNG wire#w7
   RUNG wire#powerrail
      Contact( #HMI_EXTENSION.Setup )
   END_RUNG wire#w8
   // the same network as SCL:
   "ST00310_RT01_IDB"(PLANT_IDENTIFIER := WSTRING#'+ST00310.RT01',   // "RT_2S2D1P_PD_FB"
                      ENABLE_BLOCK := "CONTROL_ON_IDB".CONTROL_ON_DELAYED_1,
                      SAFETY_OK := "IF_SAFE_TO_STND_DB".OPMode02.SafetyOK.ST00310_RT01,
                      HS_FROM_SUCCESSOR := "ST00310_DB".HS_FROM_SUCCESSOR,
                      HS_FROM_PREDECESSOR := "ST00310_DB".HS_FROM_PREDECESSOR,
                      AUTO_CONVEY_FORWARD := "ST00310_DB".VDL01.DISPLAY_INPOS2 AND ("GLOBAL_RT_2S2D1P_HMI_IF_DB".RT[23].ActData.RTDataTarget = 265),
                      AUTO_CONVEY_REVERSE := "ST00310_DB".VDL01.DISPLAY_INPOS2 AND ("GLOBAL_RT_2S2D1P_HMI_IF_DB".RT[23].ActData.RTDataTarget = 320),
                      ENABLE_FORWARD := "ST00310_DB".VDL01.DISPLAY_INPOS2 AND "ST00310_DB".FX01.DISPLAY_POS_FORWARD AND "ST00240_1_DB".LT01.POS_UP AND "OPMODE02_DB".PowerOK.ST00310_RT01_VFD01,
                      ENABLE_REVERSE := (("ST00310_DB".VDL01.DISPLAY_INPOS2 AND "ST00310_DB".FX01.DISPLAY_POS_FORWARD) OR (NOT "ST00310_DB".OPMODE.Automatic_active AND "ST00310_DB".OPMODE.Manual_active AND "ST00310_DB".VDL01.DISPLAY_INPOS1 AND "ST00310_DB".FX01.DISPLAY_POS_FORWARD)) AND "OPMODE02_DB".PowerOK.ST00310_RT01_VFD01,
                      ABS_ENABLE_FORWARD := "OPMODE02_DB".PowerOK.ST00310_VDL01_VFD01 AND NOT "ST00310_DB".VDL01_VFD01.DRIVE_RUNNING AND "OPMODE02_DB".PowerOK.ST00305_RT01_VFD01,
                      ABS_ENABLE_REVERSE := "OPMODE02_DB".PowerOK.ST00310_VDL01_VFD01 AND NOT "ST00310_DB".VDL01_VFD01.DRIVE_RUNNING,
                      PB_FORWARD := #HMI_EXTENSION.Forward,
                      PB_REVERSE := #HMI_EXTENSION.Backward,
                      POS_END_FORWARD_1 := "+ST00310.RT01-PX11:4",
                      POS_END_REVERSE := "+ST00310.RT01-PX21:4",
                      POS_SLOW_FORWARD := "+ST00310.RT01-PX12:4",
                      SELECT_FAST := #HMI_EXTENSION.Fast,
                      "RUN_W/O_ENABLE" := #HMI_EXTENSION.Setup,
                      DRIVE_READY := "ST00310_DB".RT01_VFD01.DRIVE_READY,
                      DRIVE_RUNNING := "ST00310_DB".RT01_VFD01.DRIVE_RUNNING,
                      EXTERNAL_ALARM := "ST00310_DB".Alarm,
                      SET_OCC := false,
                      OPMODE_USER_INTERFACE_OUT := "ST00310_DB".OPMODE,
                      "GLOBAL_CLOCK&SYSTEM" := "GLOBAL_INFO_IDB".HMI_GLOBAL."Clock&System",
                      IF_HMI := "GLOBAL_RT_2S2D1P_HMI_IF_DB".RT[23],
                      IF_PARA_SET := "ST00310_DB".RT01.PARA_SET,
                      HMI_SCREEN_AREA_POINTER := "GLOBAL_HMI_IF_DB".HMI_SCREEN_NO,
                      HMI_SELECT_TIMESTAMP := "GLOBAL_HMI_IF_DB".HMI_SELECT_TIMESTAMP,
                      FORWARD => "ST00310_DB".RT01.FORWARD,
                      REVERSE => "ST00310_DB".RT01.REVERSE,
                      FAST => "ST00310_DB".RT01.FAST,
                      SLOW => "ST00310_DB".RT01.SLOW,
                      JOG => "ST00310_DB".RT01.JOG,
                      OPEN_BRAKE => "ST00310_DB".RT01.OPEN_BRAKE,
                      GENERAL_ALARM => "ST00310_DB".RT01.GENERAL_ALARM,
                      HS_TO_SUCCESSOR => "ST00310_DB".RT01.HS_TO_SUCCESSOR,
                      HS_TO_PREDECESSOR => "ST00310_DB".RT01.HS_TO_PREDECESSOR,
                      DISPLAY_OCCUPIED => "ST00310_DB".RT01.DISPLAY_OCCUPIED,
                      DISPLAY_TRANSPORT => "ST00310_DB".RT01.DISPLAY_TRANSPORT,
                      DISPLAY_IN_POSITION => "ST00310_DB".RT01.DISPLAY_IN_POSITION,
                      DISPLAY_EMPTY => "ST00310_DB".RT01.DISPLAY_EMPTY,
                      DISPLAY_OCCCARBODY => "ST00310_DB".RT01.DISPLAY_OCCCARBODY,
                      DISPLAY_BLOCKENTRY => "ST00310_DB".RT01.DISPLAY_BLOCKENTRY,
                      DISPLAY_BLOCKEXIT => "ST00310_DB".RT01.DISPLAY_BLOCKEXIT);
END_REGION

REGION Network 18: RT01 Speed
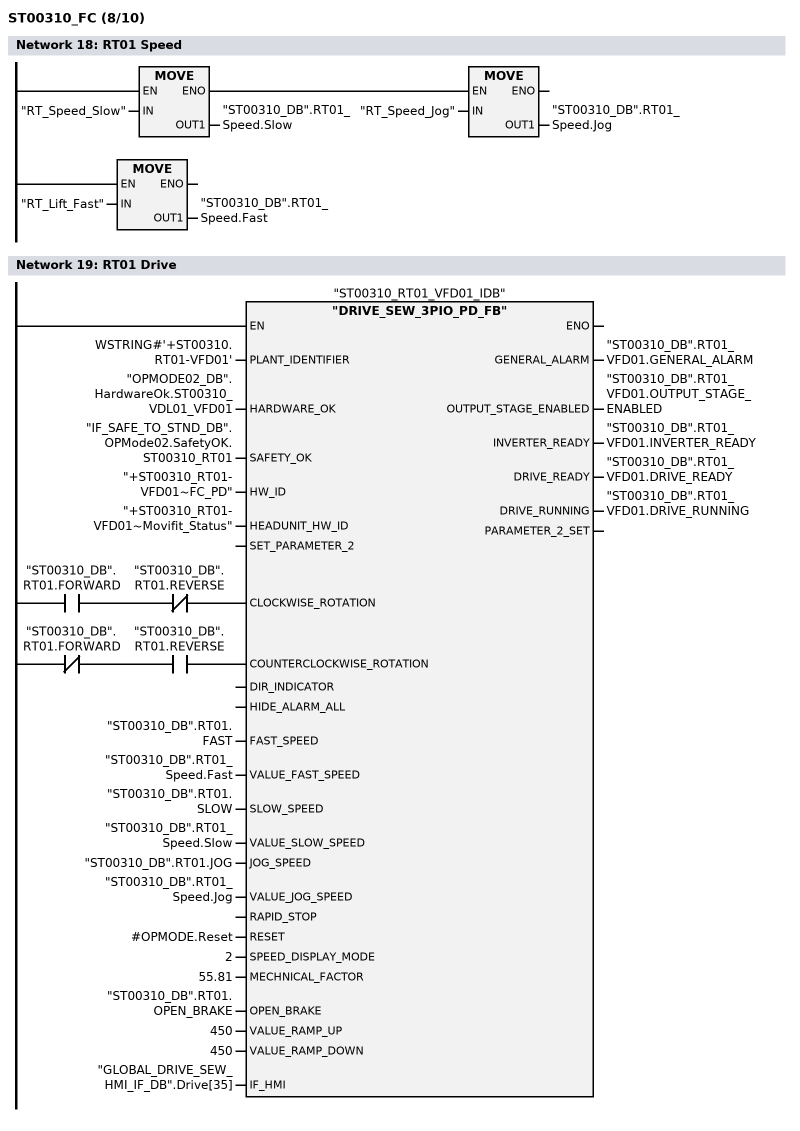
   RUNG wire#powerrail
      Move(in := "RT_Speed_Slow", out1 => "ST00310_DB".RT01_Speed.Slow)
      Move(in := "RT_Speed_Jog", out1 => "ST00310_DB".RT01_Speed.Jog)
   END_RUNG
   RUNG wire#powerrail
      Move(in := "RT_Lift_Fast", out1 => "ST00310_DB".RT01_Speed.Fast)
   END_RUNG
   // the same network as SCL:
   "ST00310_DB".RT01_Speed.Slow := "RT_Speed_Slow";
   "ST00310_DB".RT01_Speed.Jog := "RT_Speed_Jog";
   "ST00310_DB".RT01_Speed.Fast := "RT_Lift_Fast";
END_REGION

REGION Network 19: RT01 Drive
   RUNG wire#powerrail
      "ST00310_RT01_VFD01_IDB"(CLOCKWISE_ROTATION := wire#w1, COUNTERCLOCKWISE_ROTATION := wire#w2, PLANT_IDENTIFIER := WSTRING#'+ST00310.RT01-VFD01', HARDWARE_OK := "OPMODE02_DB".HardwareOk.ST00310_VDL01_VFD01, SAFETY_OK := "IF_SAFE_TO_STND_DB".OPMode02.SafetyOK.ST00310_RT01, HW_ID := "+ST00310_RT01-VFD01~FC_PD", HEADUNIT_HW_ID := "+ST00310_RT01-VFD01~Movifit_Status", SET_PARAMETER_2 :=, DIR_INDICATOR :=, HIDE_ALARM_ALL :=, FAST_SPEED := "ST00310_DB".RT01.FAST, VALUE_FAST_SPEED := "ST00310_DB".RT01_Speed.Fast, SLOW_SPEED := "ST00310_DB".RT01.SLOW, VALUE_SLOW_SPEED := "ST00310_DB".RT01_Speed.Slow, JOG_SPEED := "ST00310_DB".RT01.JOG, VALUE_JOG_SPEED := "ST00310_DB".RT01_Speed.Jog, RAPID_STOP :=, RESET := #OPMODE.Reset, SPEED_DISPLAY_MODE := 2, MECHNICAL_FACTOR := 55.81, OPEN_BRAKE := "ST00310_DB".RT01.OPEN_BRAKE, VALUE_RAMP_UP := 450, VALUE_RAMP_DOWN := 450, IF_HMI := "GLOBAL_DRIVE_SEW_HMI_IF_DB".Drive[35], GENERAL_ALARM => "ST00310_DB".RT01_VFD01.GENERAL_ALARM, OUTPUT_STAGE_ENABLED => "ST00310_DB".RT01_VFD01.OUTPUT_STAGE_ENABLED, INVERTER_READY => "ST00310_DB".RT01_VFD01.INVERTER_READY, DRIVE_READY => "ST00310_DB".RT01_VFD01.DRIVE_READY, DRIVE_RUNNING => "ST00310_DB".RT01_VFD01.DRIVE_RUNNING, PARAMETER_2_SET =>)
   END_RUNG
   RUNG wire#powerrail
      Contact( "ST00310_DB".RT01.FORWARD )
      I_Contact( "ST00310_DB".RT01.REVERSE )
   END_RUNG wire#w1
   RUNG wire#powerrail
      I_Contact( "ST00310_DB".RT01.FORWARD )
      Contact( "ST00310_DB".RT01.REVERSE )
   END_RUNG wire#w2
   // the same network as SCL:
   "ST00310_RT01_VFD01_IDB"(PLANT_IDENTIFIER := WSTRING#'+ST00310.RT01-VFD01',   // "DRIVE_SEW_3PIO_PD_FB"
                           HARDWARE_OK := "OPMODE02_DB".HardwareOk.ST00310_VDL01_VFD01,
                           SAFETY_OK := "IF_SAFE_TO_STND_DB".OPMode02.SafetyOK.ST00310_RT01,
                           HW_ID := "+ST00310_RT01-VFD01~FC_PD",
                           HEADUNIT_HW_ID := "+ST00310_RT01-VFD01~Movifit_Status",
                           CLOCKWISE_ROTATION := "ST00310_DB".RT01.FORWARD AND NOT "ST00310_DB".RT01.REVERSE,
                           COUNTERCLOCKWISE_ROTATION := NOT "ST00310_DB".RT01.FORWARD AND "ST00310_DB".RT01.REVERSE,
                           FAST_SPEED := "ST00310_DB".RT01.FAST,
                           VALUE_FAST_SPEED := "ST00310_DB".RT01_Speed.Fast,
                           SLOW_SPEED := "ST00310_DB".RT01.SLOW,
                           VALUE_SLOW_SPEED := "ST00310_DB".RT01_Speed.Slow,
                           JOG_SPEED := "ST00310_DB".RT01.JOG,
                           VALUE_JOG_SPEED := "ST00310_DB".RT01_Speed.Jog,
                           RESET := #OPMODE.Reset,
                           SPEED_DISPLAY_MODE := 2,
                           MECHNICAL_FACTOR := 55.81,
                           OPEN_BRAKE := "ST00310_DB".RT01.OPEN_BRAKE,
                           VALUE_RAMP_UP := 450,
                           VALUE_RAMP_DOWN := 450,
                           IF_HMI := "GLOBAL_DRIVE_SEW_HMI_IF_DB".Drive[35],
                           GENERAL_ALARM => "ST00310_DB".RT01_VFD01.GENERAL_ALARM,
                           OUTPUT_STAGE_ENABLED => "ST00310_DB".RT01_VFD01.OUTPUT_STAGE_ENABLED,
                           INVERTER_READY => "ST00310_DB".RT01_VFD01.INVERTER_READY,
                           DRIVE_READY => "ST00310_DB".RT01_VFD01.DRIVE_READY,
                           DRIVE_RUNNING => "ST00310_DB".RT01_VFD01.DRIVE_RUNNING);
END_REGION

REGION Network 20: *******************FX01 Control*******************
END_REGION

REGION Network 21 (SCL): FX01 Parameters
   "ST00310_DB".FX01.PARA_SET.Para.PosEndForward2 := true;
   "ST00310_DB".FX01.PARA_SET.Para.PosEndReverse2 := true;

   "ST00310_DB".FX01.PARA_SET.Set.SetRT := 100;
   "ST00310_DB".FX01.PARA_SET.Set.TimePosLeft := 20;
END_REGION

REGION Network 22: FX01 FB Control
   // To do:
   // - Add drive ready conditions
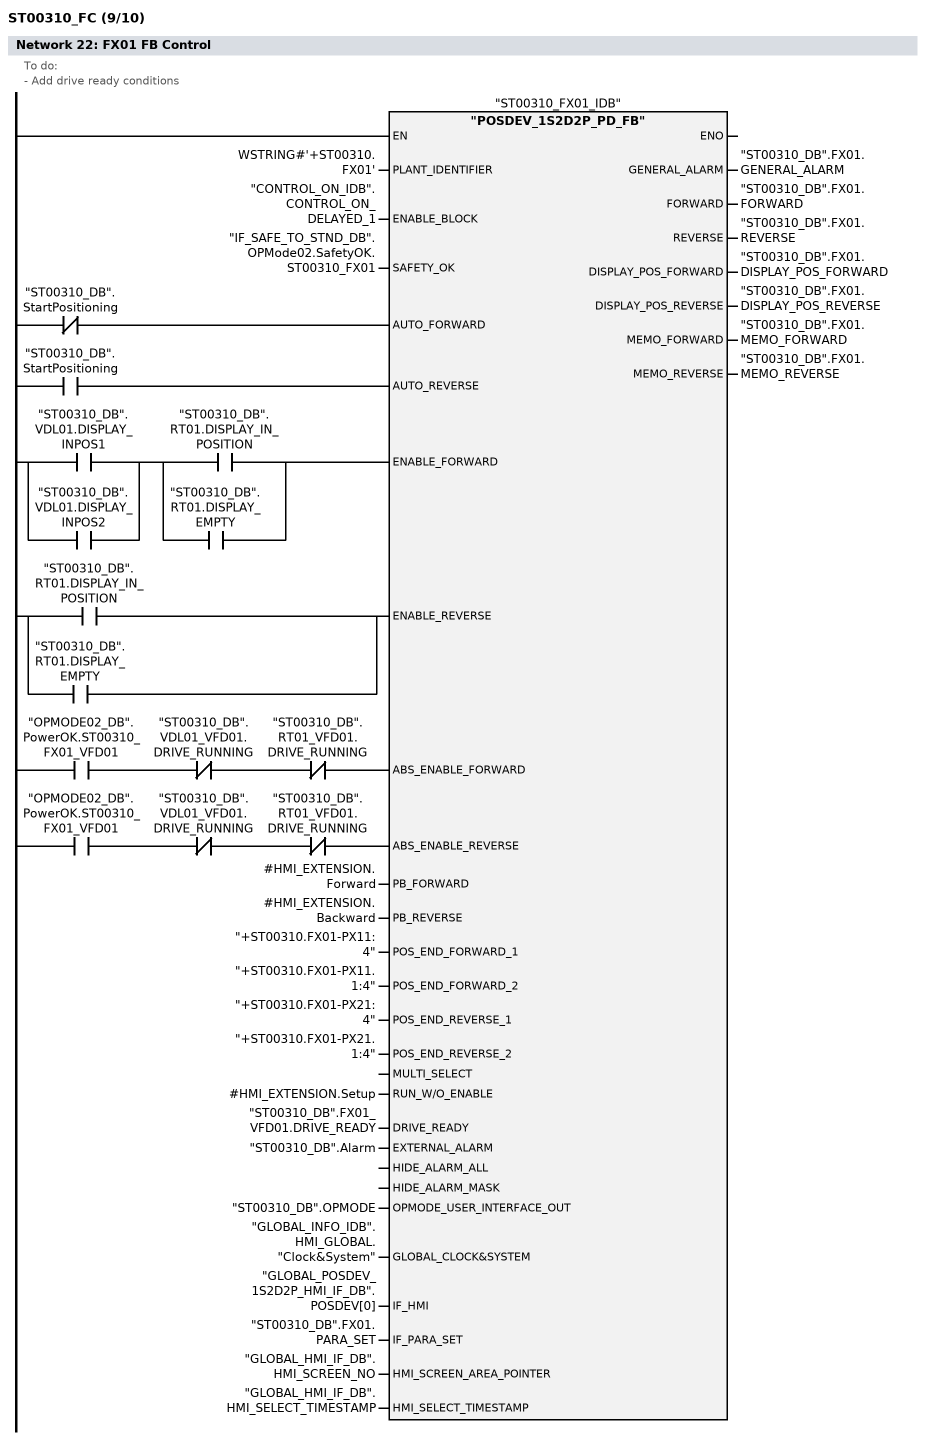
   RUNG wire#powerrail
      "ST00310_FX01_IDB"(AUTO_FORWARD := wire#w1, AUTO_REVERSE := wire#w2, ENABLE_FORWARD := wire#w4, ENABLE_REVERSE := wire#w5, ABS_ENABLE_FORWARD := wire#w6, ABS_ENABLE_REVERSE := wire#w7, PLANT_IDENTIFIER := WSTRING#'+ST00310.FX01', ENABLE_BLOCK := "CONTROL_ON_IDB".CONTROL_ON_DELAYED_1, SAFETY_OK := "IF_SAFE_TO_STND_DB".OPMode02.SafetyOK.ST00310_FX01, PB_FORWARD := #HMI_EXTENSION.Forward, PB_REVERSE := #HMI_EXTENSION.Backward, POS_END_FORWARD_1 := "+ST00310.FX01-PX11:4", POS_END_FORWARD_2 := "+ST00310.FX01-PX11.1:4", POS_END_REVERSE_1 := "+ST00310.FX01-PX21:4", POS_END_REVERSE_2 := "+ST00310.FX01-PX21.1:4", MULTI_SELECT :=, "RUN_W/O_ENABLE" := #HMI_EXTENSION.Setup, DRIVE_READY := "ST00310_DB".FX01_VFD01.DRIVE_READY, EXTERNAL_ALARM := "ST00310_DB".Alarm, HIDE_ALARM_ALL :=, HIDE_ALARM_MASK :=, OPMODE_USER_INTERFACE_OUT := "ST00310_DB".OPMODE, "GLOBAL_CLOCK&SYSTEM" := "GLOBAL_INFO_IDB".HMI_GLOBAL."Clock&System", IF_HMI := "GLOBAL_POSDEV_1S2D2P_HMI_IF_DB".POSDEV[0], IF_PARA_SET := "ST00310_DB".FX01.PARA_SET, HMI_SCREEN_AREA_POINTER := "GLOBAL_HMI_IF_DB".HMI_SCREEN_NO, HMI_SELECT_TIMESTAMP := "GLOBAL_HMI_IF_DB".HMI_SELECT_TIMESTAMP, GENERAL_ALARM => "ST00310_DB".FX01.GENERAL_ALARM, FORWARD => "ST00310_DB".FX01.FORWARD, REVERSE => "ST00310_DB".FX01.REVERSE, DISPLAY_POS_FORWARD => "ST00310_DB".FX01.DISPLAY_POS_FORWARD, DISPLAY_POS_REVERSE => "ST00310_DB".FX01.DISPLAY_POS_REVERSE, MEMO_FORWARD => "ST00310_DB".FX01.MEMO_FORWARD, MEMO_REVERSE => "ST00310_DB".FX01.MEMO_REVERSE)
   END_RUNG
   RUNG wire#powerrail
      I_Contact( "ST00310_DB".StartPositioning )
   END_RUNG wire#w1
   RUNG wire#powerrail
      Contact( "ST00310_DB".StartPositioning )
   END_RUNG wire#w2
   RUNG wire#powerrail
      Contact( "ST00310_DB".VDL01.DISPLAY_INPOS1 )
      wire#w3
      Contact( "ST00310_DB".RT01.DISPLAY_IN_POSITION )
   END_RUNG wire#w4
   RUNG wire#powerrail
      Contact( "ST00310_DB".VDL01.DISPLAY_INPOS2 )
   END_RUNG wire#w3
   RUNG wire#w3
      Contact( "ST00310_DB".RT01.DISPLAY_EMPTY )
   END_RUNG wire#w4
   RUNG wire#powerrail
      Contact( "ST00310_DB".RT01.DISPLAY_IN_POSITION )
   END_RUNG wire#w5
   RUNG wire#powerrail
      Contact( "ST00310_DB".RT01.DISPLAY_EMPTY )
   END_RUNG wire#w5
   RUNG wire#powerrail
      Contact( "OPMODE02_DB".PowerOK.ST00310_FX01_VFD01 )
      I_Contact( "ST00310_DB".VDL01_VFD01.DRIVE_RUNNING )
      I_Contact( "ST00310_DB".RT01_VFD01.DRIVE_RUNNING )
   END_RUNG wire#w6
   RUNG wire#powerrail
      Contact( "OPMODE02_DB".PowerOK.ST00310_FX01_VFD01 )
      I_Contact( "ST00310_DB".VDL01_VFD01.DRIVE_RUNNING )
      I_Contact( "ST00310_DB".RT01_VFD01.DRIVE_RUNNING )
   END_RUNG wire#w7
   // the same network as SCL:
   "ST00310_FX01_IDB"(PLANT_IDENTIFIER := WSTRING#'+ST00310.FX01',   // "POSDEV_1S2D2P_PD_FB"
                      ENABLE_BLOCK := "CONTROL_ON_IDB".CONTROL_ON_DELAYED_1,
                      SAFETY_OK := "IF_SAFE_TO_STND_DB".OPMode02.SafetyOK.ST00310_FX01,
                      AUTO_FORWARD := NOT "ST00310_DB".StartPositioning,
                      AUTO_REVERSE := "ST00310_DB".StartPositioning,
                      ENABLE_FORWARD := ("ST00310_DB".VDL01.DISPLAY_INPOS1 OR "ST00310_DB".VDL01.DISPLAY_INPOS2) AND ("ST00310_DB".RT01.DISPLAY_IN_POSITION OR "ST00310_DB".RT01.DISPLAY_EMPTY),
                      ENABLE_REVERSE := "ST00310_DB".RT01.DISPLAY_IN_POSITION OR "ST00310_DB".RT01.DISPLAY_EMPTY,
                      ABS_ENABLE_FORWARD := "OPMODE02_DB".PowerOK.ST00310_FX01_VFD01 AND NOT "ST00310_DB".VDL01_VFD01.DRIVE_RUNNING AND NOT "ST00310_DB".RT01_VFD01.DRIVE_RUNNING,
                      ABS_ENABLE_REVERSE := "OPMODE02_DB".PowerOK.ST00310_FX01_VFD01 AND NOT "ST00310_DB".VDL01_VFD01.DRIVE_RUNNING AND NOT "ST00310_DB".RT01_VFD01.DRIVE_RUNNING,
                      PB_FORWARD := #HMI_EXTENSION.Forward,
                      PB_REVERSE := #HMI_EXTENSION.Backward,
                      POS_END_FORWARD_1 := "+ST00310.FX01-PX11:4",
                      POS_END_FORWARD_2 := "+ST00310.FX01-PX11.1:4",
                      POS_END_REVERSE_1 := "+ST00310.FX01-PX21:4",
                      POS_END_REVERSE_2 := "+ST00310.FX01-PX21.1:4",
                      "RUN_W/O_ENABLE" := #HMI_EXTENSION.Setup,
                      DRIVE_READY := "ST00310_DB".FX01_VFD01.DRIVE_READY,
                      EXTERNAL_ALARM := "ST00310_DB".Alarm,
                      OPMODE_USER_INTERFACE_OUT := "ST00310_DB".OPMODE,
                      "GLOBAL_CLOCK&SYSTEM" := "GLOBAL_INFO_IDB".HMI_GLOBAL."Clock&System",
                      IF_HMI := "GLOBAL_POSDEV_1S2D2P_HMI_IF_DB".POSDEV[0],
                      IF_PARA_SET := "ST00310_DB".FX01.PARA_SET,
                      HMI_SCREEN_AREA_POINTER := "GLOBAL_HMI_IF_DB".HMI_SCREEN_NO,
                      HMI_SELECT_TIMESTAMP := "GLOBAL_HMI_IF_DB".HMI_SELECT_TIMESTAMP,
                      GENERAL_ALARM => "ST00310_DB".FX01.GENERAL_ALARM,
                      FORWARD => "ST00310_DB".FX01.FORWARD,
                      REVERSE => "ST00310_DB".FX01.REVERSE,
                      DISPLAY_POS_FORWARD => "ST00310_DB".FX01.DISPLAY_POS_FORWARD,
                      DISPLAY_POS_REVERSE => "ST00310_DB".FX01.DISPLAY_POS_REVERSE,
                      MEMO_FORWARD => "ST00310_DB".FX01.MEMO_FORWARD,
                      MEMO_REVERSE => "ST00310_DB".FX01.MEMO_REVERSE);
END_REGION

REGION Network 23: FX01 Speed
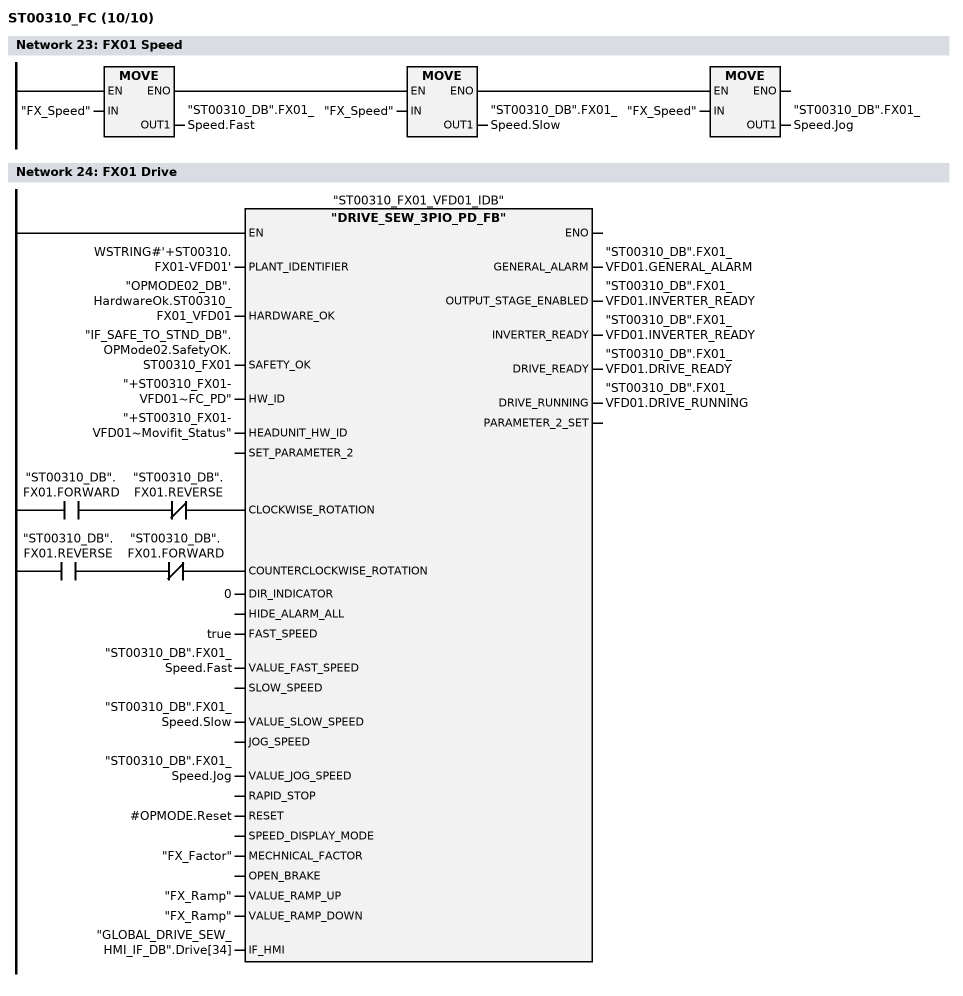
   RUNG wire#powerrail
      Move(in := "FX_Speed", out1 => "ST00310_DB".FX01_Speed.Fast)
      Move(in := "FX_Speed", out1 => "ST00310_DB".FX01_Speed.Slow)
      Move(in := "FX_Speed", out1 => "ST00310_DB".FX01_Speed.Jog)
   END_RUNG
   // the same network as SCL:
   "ST00310_DB".FX01_Speed.Fast := "FX_Speed";
   "ST00310_DB".FX01_Speed.Slow := "FX_Speed";
   "ST00310_DB".FX01_Speed.Jog := "FX_Speed";
END_REGION

REGION Network 24: FX01 Drive
   RUNG wire#powerrail
      "ST00310_FX01_VFD01_IDB"(CLOCKWISE_ROTATION := wire#w1, COUNTERCLOCKWISE_ROTATION := wire#w2, PLANT_IDENTIFIER := WSTRING#'+ST00310.FX01-VFD01', HARDWARE_OK := "OPMODE02_DB".HardwareOk.ST00310_FX01_VFD01, SAFETY_OK := "IF_SAFE_TO_STND_DB".OPMode02.SafetyOK.ST00310_FX01, HW_ID := "+ST00310_FX01-VFD01~FC_PD", HEADUNIT_HW_ID := "+ST00310_FX01-VFD01~Movifit_Status", SET_PARAMETER_2 :=, DIR_INDICATOR := 0, HIDE_ALARM_ALL :=, FAST_SPEED := true, VALUE_FAST_SPEED := "ST00310_DB".FX01_Speed.Fast, SLOW_SPEED :=, VALUE_SLOW_SPEED := "ST00310_DB".FX01_Speed.Slow, JOG_SPEED :=, VALUE_JOG_SPEED := "ST00310_DB".FX01_Speed.Jog, RAPID_STOP :=, RESET := #OPMODE.Reset, SPEED_DISPLAY_MODE :=, MECHNICAL_FACTOR := "FX_Factor", OPEN_BRAKE :=, VALUE_RAMP_UP := "FX_Ramp", VALUE_RAMP_DOWN := "FX_Ramp", IF_HMI := "GLOBAL_DRIVE_SEW_HMI_IF_DB".Drive[34], GENERAL_ALARM => "ST00310_DB".FX01_VFD01.GENERAL_ALARM, OUTPUT_STAGE_ENABLED => "ST00310_DB".FX01_VFD01.INVERTER_READY, INVERTER_READY => "ST00310_DB".FX01_VFD01.INVERTER_READY, DRIVE_READY => "ST00310_DB".FX01_VFD01.DRIVE_READY, DRIVE_RUNNING => "ST00310_DB".FX01_VFD01.DRIVE_RUNNING, PARAMETER_2_SET =>)
   END_RUNG
   RUNG wire#powerrail
      Contact( "ST00310_DB".FX01.FORWARD )
      I_Contact( "ST00310_DB".FX01.REVERSE )
   END_RUNG wire#w1
   RUNG wire#powerrail
      Contact( "ST00310_DB".FX01.REVERSE )
      I_Contact( "ST00310_DB".FX01.FORWARD )
   END_RUNG wire#w2
   // the same network as SCL:
   "ST00310_FX01_VFD01_IDB"(PLANT_IDENTIFIER := WSTRING#'+ST00310.FX01-VFD01',   // "DRIVE_SEW_3PIO_PD_FB"
                           HARDWARE_OK := "OPMODE02_DB".HardwareOk.ST00310_FX01_VFD01,
                           SAFETY_OK := "IF_SAFE_TO_STND_DB".OPMode02.SafetyOK.ST00310_FX01,
                           HW_ID := "+ST00310_FX01-VFD01~FC_PD",
                           HEADUNIT_HW_ID := "+ST00310_FX01-VFD01~Movifit_Status",
                           CLOCKWISE_ROTATION := "ST00310_DB".FX01.FORWARD AND NOT "ST00310_DB".FX01.REVERSE,
                           COUNTERCLOCKWISE_ROTATION := "ST00310_DB".FX01.REVERSE AND NOT "ST00310_DB".FX01.FORWARD,
                           DIR_INDICATOR := 0,
                           FAST_SPEED := true,
                           VALUE_FAST_SPEED := "ST00310_DB".FX01_Speed.Fast,
                           VALUE_SLOW_SPEED := "ST00310_DB".FX01_Speed.Slow,
                           VALUE_JOG_SPEED := "ST00310_DB".FX01_Speed.Jog,
                           RESET := #OPMODE.Reset,
                           MECHNICAL_FACTOR := "FX_Factor",
                           VALUE_RAMP_UP := "FX_Ramp",
                           VALUE_RAMP_DOWN := "FX_Ramp",
                           IF_HMI := "GLOBAL_DRIVE_SEW_HMI_IF_DB".Drive[34],
                           GENERAL_ALARM => "ST00310_DB".FX01_VFD01.GENERAL_ALARM,
                           OUTPUT_STAGE_ENABLED => "ST00310_DB".FX01_VFD01.INVERTER_READY,
                           INVERTER_READY => "ST00310_DB".FX01_VFD01.INVERTER_READY,
                           DRIVE_READY => "ST00310_DB".FX01_VFD01.DRIVE_READY,
                           DRIVE_RUNNING => "ST00310_DB".FX01_VFD01.DRIVE_RUNNING);
END_REGION
END_FUNCTION
